FUNCTION_BLOCK Skill_PickPlace  EXTENDS FB_1_Skill
// FB_2_Skill_SFC
VAR_INPUT
	pRob: POINTER TO FB_2_ROB_MANIP;
	{attribute 'OPC.UA.DA.StructuredType':=1}
	{attribute 'OPC.UA.DA' := '1'}
	Param: POINTER TO stParam_PickPlace;
	SFCInit: BOOL;
END_VAR
VAR_OUTPUT
	
END_VAR
VAR
	approachpick, approachplace,pickpos,placepos : ST_Pose;


	

	res: eResult;
	bCalcApproachDone: BOOL;
	phase: INT;

	Settings: stCommand_Settings;

	bMoveInProcess: BOOL;
	bMovePickApproachDone: BOOL;
	bMovePickDone: BOOL;
	runningSkill: POINTER TO FB_1_Skill;
	bGripperCloseDone: BOOL;
	bRetractPickDone: BOOL;
	bMovePlaceApproachDone: BOOL;
	bMovePlaceDone: BOOL;
	bGripperOpenDone: BOOL;
	bRetractPlaceDone: BOOL;
	middlepoint: ST_Pose;
	bGotMiddlePoint: BOOL;
	bveMiddlePointDone: BOOL;
	bMoveMiddlePointDone: BOOL;
	T_Point: ST_TransformMatrix;
	
	T_Offset: ST_TransformMatrix;
	T_Result: ST_TransformMatrix;
END_VAR

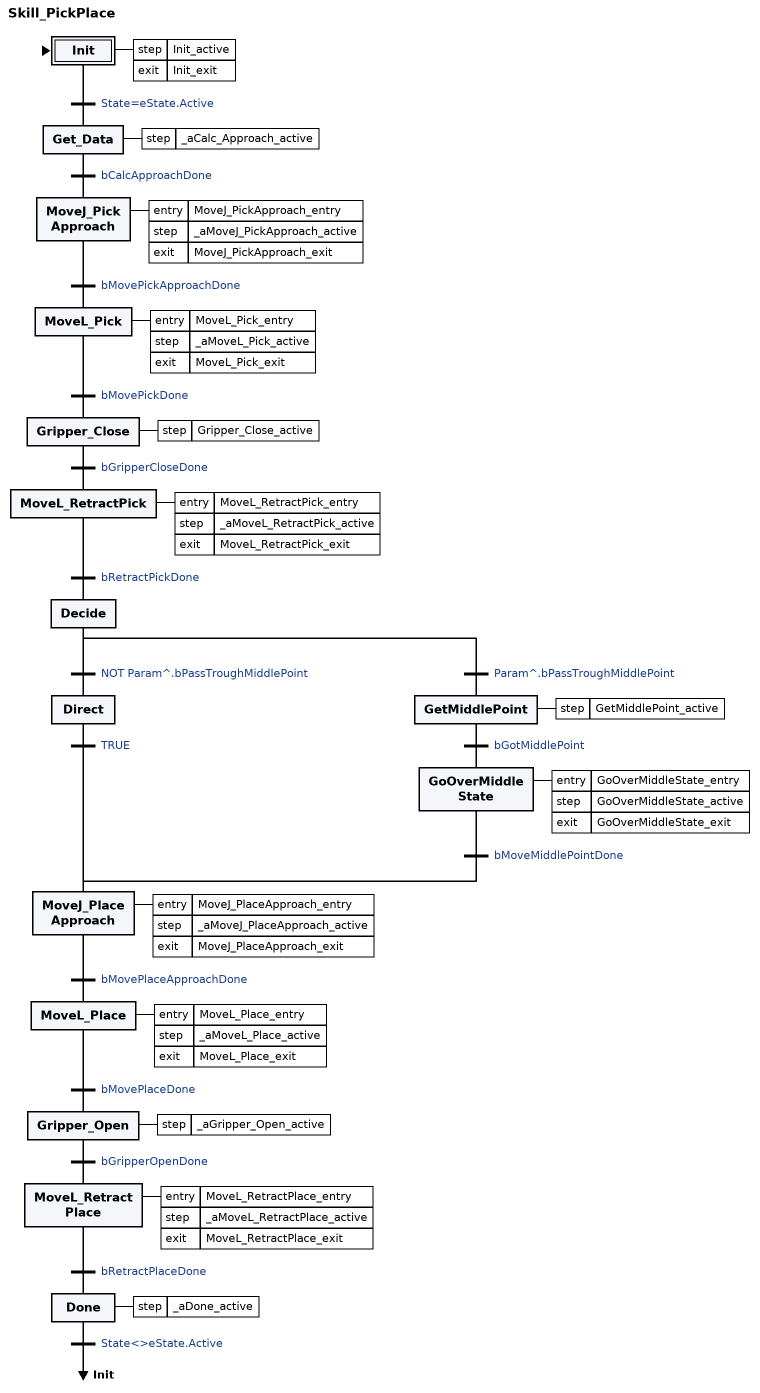
INITIAL_STEP Init:
    Init_active(N);  // step action
    Init_exit(P0);  // exit action
END_STEP
TRANSITION FROM Init TO Get_Data
    := State=eState.Active;
END_TRANSITION
STEP Get_Data:
    _aCalc_Approach_active(N);  // step action
END_STEP
TRANSITION FROM Get_Data TO MoveJ_PickApproach
    := bCalcApproachDone;
END_TRANSITION
STEP MoveJ_PickApproach:
    MoveJ_PickApproach_entry(P1);  // entry action
    _aMoveJ_PickApproach_active(N);  // step action
    MoveJ_PickApproach_exit(P0);  // exit action
END_STEP
TRANSITION FROM MoveJ_PickApproach TO MoveL_Pick
    := bMovePickApproachDone;
END_TRANSITION
STEP MoveL_Pick:
    MoveL_Pick_entry(P1);  // entry action
    _aMoveL_Pick_active(N);  // step action
    MoveL_Pick_exit(P0);  // exit action
END_STEP
TRANSITION FROM MoveL_Pick TO Gripper_Close
    := bMovePickDone;
END_TRANSITION
STEP Gripper_Close:
    Gripper_Close_active(N);  // step action
END_STEP
TRANSITION FROM Gripper_Close TO MoveL_RetractPick
    := bGripperCloseDone;
END_TRANSITION
STEP MoveL_RetractPick:
    MoveL_RetractPick_entry(P1);  // entry action
    _aMoveL_RetractPick_active(N);  // step action
    MoveL_RetractPick_exit(P0);  // exit action
END_STEP
TRANSITION FROM MoveL_RetractPick TO Decide
    := bRetractPickDone;
END_TRANSITION
STEP Decide:
END_STEP
TRANSITION FROM Decide TO Direct
    := NOT Param^.bPassTroughMiddlePoint;
END_TRANSITION
STEP Direct:
END_STEP
TRANSITION FROM Direct TO MoveJ_PlaceApproach
    := TRUE;
END_TRANSITION
TRANSITION FROM Decide TO GetMiddlePoint
    := Param^.bPassTroughMiddlePoint;
END_TRANSITION
STEP GetMiddlePoint:
    GetMiddlePoint_active(N);  // step action
END_STEP
TRANSITION FROM GetMiddlePoint TO GoOverMiddleState
    := bGotMiddlePoint;
END_TRANSITION
STEP GoOverMiddleState:
    GoOverMiddleState_entry(P1);  // entry action
    GoOverMiddleState_active(N);  // step action
    GoOverMiddleState_exit(P0);  // exit action
END_STEP
TRANSITION FROM GoOverMiddleState TO MoveJ_PlaceApproach
    := bMoveMiddlePointDone;
END_TRANSITION
STEP MoveJ_PlaceApproach:
    MoveJ_PlaceApproach_entry(P1);  // entry action
    _aMoveJ_PlaceApproach_active(N);  // step action
    MoveJ_PlaceApproach_exit(P0);  // exit action
END_STEP
TRANSITION FROM MoveJ_PlaceApproach TO MoveL_Place
    := bMovePlaceApproachDone;
END_TRANSITION
STEP MoveL_Place:
    MoveL_Place_entry(P1);  // entry action
    _aMoveL_Place_active(N);  // step action
    MoveL_Place_exit(P0);  // exit action
END_STEP
TRANSITION FROM MoveL_Place TO Gripper_Open
    := bMovePlaceDone;
END_TRANSITION
STEP Gripper_Open:
    _aGripper_Open_active(N);  // step action
END_STEP
TRANSITION FROM Gripper_Open TO MoveL_RetractPlace
    := bGripperOpenDone;
END_TRANSITION
STEP MoveL_RetractPlace:
    MoveL_RetractPlace_entry(P1);  // entry action
    _aMoveL_RetractPlace_active(N);  // step action
    MoveL_RetractPlace_exit(P0);  // exit action
END_STEP
TRANSITION FROM MoveL_RetractPlace TO Done
    := bRetractPlaceDone;
END_TRANSITION
STEP Done:
    _aDone_active(N);  // step action
END_STEP
TRANSITION FROM Done TO Init
    := State<>eState.Active;
END_TRANSITION

ACTION _aCalc_Approach_active:
// TODO: Resolve Param.PickPositionName / Param.PlacePositionName to base poses.
// Apply PickPositionOffset / PlacePositionOffset and calculate approachpick / approachplace
// from PickApproachDirection / PlaceApproachDirection and the configured offsets.
// Set bCalcApproachDone := TRUE when both poses are valid.

IF phase = 0 THEN
	IF Param^.PickPositionName<>'' THEN
		res := pRob^.PM.Load(Param^.PickPositionName);
		
		IF res=SUCCESS THEN
			T_Point  := FromPose(pRob^.PM.LoadedPose);
			T_Offset := FromPose(Param^.PickPositionOffset);
			
			T_Result := Multiply(
				A := T_Point,
				B := T_Offset
			);
			
			pickpos := ToPose(T_Result);
			phase := 10;
		ELSE
			ExecutionDone:=TRUE;
			ExecutionResult:=FAILURE;
			Deactivate();
			Messenger.AddError(eMessageCategories.MissingData,Path,'Pick Position is not defined in PM');
			SFCInit:=TRUE;
			
		END_IF
	END_IF
END_IF


IF phase = 10 THEN
	IF Param^.PlacePositionName<>'' THEN
		res := pRob^.PM.Load(Param^.PlacePositionName);
		
		IF res=SUCCESS THEN
      placepos := pROB^.PM.LoadedPose;
      placepos.x := placepos.x + Param^.PlacePositionOffset.x;
      placepos.y := placepos.y + Param^.PlacePositionOffset.y;
      placepos.z := placepos.z + Param^.PlacePositionOffset.z;
      placepos.roll := placepos.roll + Param^.PlacePositionOffset.roll;
      placepos.pitch := placepos.pitch + Param^.PlacePositionOffset.pitch;
      placepos.yaw := placepos.yaw + Param^.PlacePositionOffset.yaw;
			phase := 20;
		ELSE
			ExecutionDone:=TRUE;
			ExecutionResult:=FAILURE;
			Deactivate();
			Messenger.AddError(eMessageCategories.MissingData,Path,'Place Position is not defined in PM');
			SFCInit:=TRUE;
			
		END_IF
	END_IF
END_IF



IF phase = 20 THEN
	approachpick := F_CalcOffsetPose(pickpos,Param^.PickApproachDirection,Param^.PickApproachOffset);
	approachplace := F_CalcOffsetPose(placepos,Param^.PlaceApproachDirection,Param^.PlaceApproachOffset);
	bCalcApproachDone := TRUE;
END_IF
END_ACTION

ACTION _aDone_active:
ExecutionDone:=TRUE;
ExecutionResult:=SUCCESS;
END_ACTION

ACTION _aGripper_Close_active:

END_ACTION

ACTION _aGripper_Open_active:
IF pRob^.TOOL^.Release() = SUCCESS THEN
	bGripperOpenDone:=TRUE;
END_IF
END_ACTION

ACTION _aMoveJ_PickApproach_active:
PollRobotMove(DoneFlag := bMovePickApproachDone);
END_ACTION

ACTION _aMoveJ_PlaceApproach_active:
PollRobotMove(DoneFlag := bMovePlaceApproachDone);
END_ACTION

ACTION _aMoveL_Pick_active:
PollRobotMove(DoneFlag := bMovePickDone);
END_ACTION

ACTION _aMoveL_Place_active:
PollRobotMove(DoneFlag := bMovePlaceDone);
END_ACTION

ACTION _aMoveL_RetractPick_active:
PollRobotMove(DoneFlag := bRetractPickDone);
END_ACTION

ACTION _aMoveL_RetractPlace_active:
PollRobotMove(DoneFlag := bRetractPlaceDone);
END_ACTION

ACTION GetMiddlePoint_active:
// TODO: Resolve Param.PickPositionName / Param.PlacePositionName to base poses.
// Apply PickPositionOffset / PlacePositionOffset and calculate approachpick / approachplace
// from PickApproachDirection / PlaceApproachDirection and the configured offsets.
// Set bCalcApproachDone := TRUE when both poses are valid.

IF Param^.MiddlePointName<>'' THEN
	res := pRob^.PM.Load(Param^.MiddlePointName);
	
	IF res=SUCCESS THEN
		middlepoint := pROB^.PM.LoadedPose;
		bGotMiddlePoint := TRUE;
	END_IF
END_IF
END_ACTION

ACTION GoOverMiddleState_active:
PollRobotMove(DoneFlag := bMoveMiddlePointDone);
END_ACTION

ACTION GoOverMiddleState_entry:
Settings.Target.pose:=middlepoint;
Settings.Target.frame_id:= eRefFrame.BRF;
Settings.Velocity:=Param^.FastVelocity;


nCalledCmdID := pRob^.MoveJoint(
  Target := Settings.Target,
  Velocity := Param^.FastVelocity);
HandleMoveStart();
END_ACTION

ACTION GoOverMiddleState_exit:
nCalledCmdID:=0;
bMoveInProcess:=FALSE;
bMoveMiddlePointDone:=FALSE;
END_ACTION

ACTION Gripper_Close_active:
IF pRob^.TOOL^.Grip() = SUCCESS THEN
	bGripperCloseDone:=TRUE;
END_IF
END_ACTION

ACTION Gripper_Close_entry:

END_ACTION

ACTION Gripper_Close_exit:
bSubSkillRunning:=FALSE;
END_ACTION

METHOD HandleMoveStart : BOOL
HandleMoveStart := nCalledCmdID <> 0;

  IF NOT HandleMoveStart THEN
      ExecutionDone := TRUE;
      ExecutionResult := FAILURE;
      Messenger.AddWarn(eMessageCategories.ParentFailed, Path, 'Robot rejected move');
      SFCInit := TRUE;
  END_IF
END_METHOD

ACTION Init_active:
phase:=0;
nCalledCmdID := 0;
bMoveInProcess := FALSE;

bMovePickApproachDone	:=FALSE;
bMovePickDone			:=FALSE;
bGripperCloseDone		:=FALSE;
bRetractPickDone		:=FALSE;
bMovePlaceApproachDone	:=FALSE;
bMovePlaceDone			:=FALSE;
bGripperOpenDone		:=FALSE;
bRetractPlaceDone		:=FALSE;
bGotMiddlePoint			:=FALSE;
bveMiddlePointDone		:=FALSE;
bMoveMiddlePointDone	:=FALSE;
END_ACTION

ACTION Init_exit:
ExecutionDone:=FALSE;
ExecutionResult:=NONE;

phase:=0;
nCalledCmdID := 0;
bMoveInProcess := FALSE;

bMovePickApproachDone	:=FALSE;
bMovePickDone			:=FALSE;
bGripperCloseDone		:=FALSE;
bRetractPickDone		:=FALSE;
bMovePlaceApproachDone	:=FALSE;
bMovePlaceDone			:=FALSE;
bGripperOpenDone		:=FALSE;
bRetractPlaceDone		:=FALSE;
bGotMiddlePoint			:=FALSE;
bveMiddlePointDone		:=FALSE;
bMoveMiddlePointDone	:=FALSE;
END_ACTION

ACTION MoveJ_PickApproach_entry:
bCalcApproachDone:=FALSE;


Settings.Target.pose:=approachpick;
Settings.Target.frame_id:= eRefFrame.BRF;
Settings.Velocity:=Param^.FastVelocity;


nCalledCmdID := pRob^.MoveJoint(
  Target := Settings.Target,
  Velocity := Param^.FastVelocity);
HandleMoveStart();
END_ACTION

ACTION MoveJ_PickApproach_exit:
nCalledCmdID:=0;
bMoveInProcess:=FALSE;
bMovePickApproachDone := FALSE;
END_ACTION

ACTION MoveJ_PlaceApproach_entry:
Settings.Target.pose:=approachplace;
Settings.Target.frame_id:= eRefFrame.BRF;

Settings.Velocity:=Param^.FastVelocity;


nCalledCmdID := pRob^.MoveJoint(
  Target := Settings.Target,
  Velocity := Param^.FastVelocity);
HandleMoveStart();
END_ACTION

ACTION MoveJ_PlaceApproach_exit:
nCalledCmdID:=0;
bMoveInProcess:=FALSE;
bMovePlaceApproachDone := FALSE;
END_ACTION

ACTION MoveL_Pick_entry:


Settings.Target.pose:=pickpos;
Settings.Target.frame_id:= eRefFrame.BRF;
Settings.Velocity:=Param^.SlowVelocity;


nCalledCmdID := pRob^.MoveLinear(
  Target := Settings.Target,
  Velocity := Param^.SlowVelocity);
HandleMoveStart();
END_ACTION

ACTION MoveL_Pick_exit:
nCalledCmdID:=0;
bMoveInProcess:=FALSE;
bMovePickDone := FALSE;
END_ACTION

ACTION MoveL_Place_entry:
Settings.Target.pose:=placepos;
Settings.Target.frame_id:= eRefFrame.BRF;

Settings.Velocity:=Param^.SlowVelocity;


nCalledCmdID := pRob^.MoveLinear(
  Target := Settings.Target,
  Velocity := Param^.SlowVelocity);
HandleMoveStart();
END_ACTION

ACTION MoveL_Place_exit:
nCalledCmdID:=0;
bMoveInProcess:=FALSE;
bMovePlaceDone := FALSE;
END_ACTION

ACTION MoveL_RetractPick_entry:
Settings.Target.pose:=approachpick;
Settings.Target.frame_id:= eRefFrame.BRF;
Settings.Velocity:=Param^.SlowVelocity;


nCalledCmdID := pRob^.MoveLinear(
  Target := Settings.Target,
  Velocity := Param^.SlowVelocity);
HandleMoveStart();
END_ACTION

ACTION MoveL_RetractPick_exit:
nCalledCmdID:=0;
bMoveInProcess:=FALSE;
bRetractPickDone := FALSE;
END_ACTION

ACTION MoveL_RetractPlace_entry:
Settings.Target.pose:=approachplace;
Settings.Target.frame_id:= eRefFrame.BRF;

Settings.Velocity:=Param^.SlowVelocity;


nCalledCmdID := pRob^.MoveLinear(
  Target := Settings.Target,
  Velocity := Param^.SlowVelocity);
HandleMoveStart();
END_ACTION

ACTION MoveL_RetractPlace_exit:
nCalledCmdID:=0;
bMoveInProcess:=FALSE;
bRetractPlaceDone := FALSE;
END_ACTION

METHOD PROTECTED OnActivate : eResult
VAR_INPUT
END_VAR

VAR
	eParentResult: eResult;
	myResult: ERESULT;
END_VAR

VAR //YOUR CODE
	succ : BOOL;
END_VAR
eParentResult := SUPER^.OnActivate();
//--------------------------------------------------
myResult:=NONE;
// ----- YOUR CODE HERE (incl. Alarms) -------------

SFCInit:=FALSE;
myResult:=SUCCESS;



// ----- END YOUR CODE -----------------------------
//--------------------------------------------------
OnActivate := CombineResults(eParentResult,myResult);
END_METHOD

METHOD PROTECTED OnDeactivate : eResult
VAR_INPUT
END_VAR

VAR
	eParentResult: eResult;
	myResult: ERESULT;
END_VAR

VAR //YOUR CODE
	succ : BOOL;
END_VAR
eParentResult := SUPER^.OnDeactivate();
//--------------------------------------------------
myResult:=NONE;
// ----- YOUR CODE HERE (incl. Alarms) -------------

SFCInit:=TRUE;
myResult:=SUCCESS;
bMoveInProcess:=FALSE;

// ----- END YOUR CODE -----------------------------
//--------------------------------------------------
OnDeactivate := CombineResults(eParentResult,myResult);
END_METHOD

METHOD PROTECTED OnError : eResult
VAR_INPUT
END_VAR

VAR
	eParentResult: eResult;
	myResult: ERESULT;
END_VAR

VAR //YOUR CODE
	succ : BOOL;
END_VAR
eParentResult := SUPER^.OnError();

myResult := NONE;

// ----- YOUR CODE HERE -----------------------------
SFCInit:=TRUE;
myResult := SUCCESS;

// ----- END YOUR CODE ------------------------------

OnError := CombineResults(eParentResult, myResult);
END_METHOD

METHOD PROTECTED OnShutdown : eResult
VAR_INPUT
END_VAR

    VAR
    	eParentResult: eResult;
    	myResult: ERESULT;
    END_VAR

    VAR //YOUR CODE
    	succ : BOOL;
    END_VAR
eParentResult := SUPER^.OnShutdown();
//--------------------------------------------------
myResult:=NONE;
// ----- YOUR CODE HERE (incl. Alarms) -------------


SFCInit:=TRUE;
myResult:=SUCCESS;

// ----- END YOUR CODE -----------------------------
//--------------------------------------------------
OnShutdown := CombineResults(eParentResult,myResult);
END_METHOD

METHOD PollRobotMove : BOOL
    VAR_IN_OUT
      DoneFlag : BOOL;
    END_VAR
PollRobotMove := FALSE;

    IF pRob = 0 THEN
      ExecutionDone := TRUE;
      ExecutionResult := ERROR;
      Messenger.AddError(eMessageCategories.MissingData, Path, 'Robot is not assigned');
      SFCInit := TRUE;
      RETURN;
    END_IF

    IF (nCalledCmdID = 0) OR (pRob^.CommandID <> nCalledCmdID) THEN
      RETURN;
    END_IF

    bMoveInProcess := TRUE;

    CASE pRob^.CommandState OF
      eProgress.INIT, eProgress.ACKNOWLEDGE, eProgress.RUNNING:
        PollRobotMove := FALSE;

      eProgress.FINALIZED:
        IF pRob^.CommandResult = SUCCESS THEN
          DoneFlag := TRUE;
          PollRobotMove := TRUE;
        ELSE
          ExecutionDone := TRUE;
          IF pRob^.CommandResult = NONE THEN
            ExecutionResult := ERROR;
          ELSE
            ExecutionResult := pRob^.CommandResult;
          END_IF
          Messenger.AddWarn(eMessageCategories.ParentFailed, Path, 'Robot move failed');
          SFCInit := TRUE;
        END_IF

      eProgress.ABORTED:
        ExecutionDone := TRUE;
        ExecutionResult := FAILURE;
        Messenger.AddWarn(eMessageCategories.ParentFailed, Path, 'Robot move aborted');
        SFCInit := TRUE;
    END_CASE
END_METHOD

END_FUNCTION_BLOCK

(* stored: Version 1.1.0.1, ProductVersion 3.1.4026.18
   POU Skill_PickPlace: Id {19f0d2dc-4f3e-4476-b186-4f85a96e59fa}, SpecialFunc None
   Folder StateControl: Id {b8625484-5b9d-403b-b98f-c4de5899beed}
   Action _aCalc_Approach_active: Id {37dfacd0-5ddb-427e-a6d5-ffb024477c13}
   Action _aDone_active: Id {e89f9719-0119-4542-a78a-a5b9a7f93659}
   Action _aGripper_Close_active: Id {9ee85894-a04e-49cb-9fef-a6b3351f6680}
   Action _aGripper_Open_active: Id {cf90c9f8-9efe-4b16-b87d-425e4fed125f}
   Action _aMoveJ_PickApproach_active: Id {92d00584-9814-4e39-8fa3-8493e89622e3}
   Action _aMoveJ_PlaceApproach_active: Id {a42b9b23-6938-4b16-8ea5-134746ad2288}
   Action _aMoveL_Pick_active: Id {73b9f592-c1d9-4003-92ee-e278bc29956d}
   Action _aMoveL_Place_active: Id {2c5e09cd-59b9-42e3-be17-fb01c6d6beaf}
   Action _aMoveL_RetractPick_active: Id {cffa91e5-3624-4087-864a-9d66af7cbc22}
   Action _aMoveL_RetractPlace_active: Id {7ddb2123-18b0-4656-a4f2-c9374296db50}
   Action GetMiddlePoint_active: Id {f4d50aa2-832a-4fa3-a8a2-72d5c28f6d4c}
   Action GoOverMiddleState_active: Id {7db3ba8f-331b-4fb1-bdef-854308e83b1d}
   Action GoOverMiddleState_entry: Id {26f5b4c1-e04f-4111-8bad-0c088371fe18}
   Action GoOverMiddleState_exit: Id {c627f6fa-cc85-4a31-8f6e-63da895398bc}
   Action Gripper_Close_active: Id {b462e5a3-d3e4-40a1-b1d0-970ba279ea7b}
   Action Gripper_Close_entry: Id {dfa66bf6-7f5b-4a42-b3f9-0a95de0f88f9}
   Action Gripper_Close_exit: Id {1a37bfea-119a-434a-994d-1e022c907901}
   Method HandleMoveStart: Id {57dbf99b-ec72-47c9-a087-a8267dfa732e}
   Action Init_active: Id {bb9d285b-87dd-4209-82d5-a350113088c8}
   Action Init_exit: Id {d8ae8678-7787-4082-8e7b-633a4307d317}
   Action MoveJ_PickApproach_entry: Id {81ae2925-3ee5-40ec-bd66-01c408ed70f4}
   Action MoveJ_PickApproach_exit: Id {e2f5d488-d4c7-4a0e-a42e-a26a64f7b9c5}
   Action MoveJ_PlaceApproach_entry: Id {832e16b5-ffc9-47bb-8153-73fd53b7df55}
   Action MoveJ_PlaceApproach_exit: Id {5229f4b1-1f3d-4f1d-bbe3-c51f7e0fb745}
   Action MoveL_Pick_entry: Id {0cdfa23a-60a7-423e-9402-9b391ce28731}
   Action MoveL_Pick_exit: Id {73135b79-08b7-4530-8720-be518dca25f8}
   Action MoveL_Place_entry: Id {a4302577-19dd-47de-9f54-8cd72711ffe8}
   Action MoveL_Place_exit: Id {84a61dec-1718-453c-a818-66168ad7e659}
   Action MoveL_RetractPick_entry: Id {17e20099-1738-4082-955e-656ad5d96d34}
   Action MoveL_RetractPick_exit: Id {a05a6f6a-3c5c-4092-86c8-c0c55643a997}
   Action MoveL_RetractPlace_entry: Id {48b6db56-5e1b-4e06-960d-59187aa3853a}
   Action MoveL_RetractPlace_exit: Id {5c7fa900-9614-4520-a58b-fa98fb8c9bc2}
   Method OnActivate: Id {fe361160-cff6-4374-b8d5-b6aa8065f810}
   Method OnDeactivate: Id {b3c5dbd6-4410-45d6-8fa7-b9583ee78948}
   Method OnError: Id {399d5806-abb9-4580-87f6-befc1c718003}
   Method OnShutdown: Id {8cf91fc1-76e2-44cf-a181-f40f308b193c}
   Method PollRobotMove: Id {78fd90e9-ae41-49ae-a2ac-70ab9188a9db} *)
